// SIMATIC STEP 7 (V5.x) project Kukla-DP-DWC7A
// CPU: CPU 315-2 PN/DP
// station: Hardware
// station: SIMATIC 300(1)
// station: P_ADR_BUS
// program: S7 Prog DWC7A

SYMBOL_TABLE
"CMD_KSW"	DB 40	DB 40
"ACT_KSW"	DB 41	DB 41	// Datablock for Continious weighing system 1
"COMM_KSW7"	FC 40	FC 40
"PLC_toKSW7B"	VAT 1		// DB40_PLC_to_KSW
"KSW7B_to_PLC"	VAT 2		// DB41_KSW7_to_PLC
END_SYMBOL_TABLE

TYPE UDT 400
VERSION : 1.0
  STRUCT
   bWCx_Warning : BOOL ;	// 24: Warnung
   bWCx_RdyToOperate : BOOL ;	// 25: Betriebsbereit
   bWCx_XD0 : BOOL ;	// 26:
   bWCx_XD1 : BOOL ;	// 27:
   bWCx_XD2 : BOOL ;	// 28:
   bWCx_XD3 : BOOL ;	// 29:
   bWCx_Crtl_30 : BOOL ;	// 30: ---
   bWCx_FieldRelais4 : BOOL ;	// 31: Fieldrelais 4
   bWCx_DriveBolcked : BOOL ;	// 16: Antriebe gesperrt
   bWCx_EmcyStopActiv : BOOL ;	// 17: Notaus aktiv
   bWCx_MainDriveRuns : BOOL ;	// 18: Läuft
   bWCx_MainDriveJog : BOOL ;	// 19: Hauptantrieb JOG
   bWCx_FieldRelais0 : BOOL ;	// 20: Fieldrelais 0
   bWCx_FieldRelais1 : BOOL ;	// 21: Fieldrelais 1
   bWCx_FieldRelais2 : BOOL ;	// 22: Fieldrelais 2
   bWCx_FieldRelais3 : BOOL ;	// 23: Fieldrelais 3
   bWCx_BinMaxLevel : BOOL ;	// 08: Max Meldung
   bWCx_BinMaxMaxLevel : BOOL ;	// 09: Max Max Meldung
   bWCx_BatchWeightFault : BOOL ;	// 10: Mengenfehler
   bWCx_Crtl_11 : BOOL ;	// 11: ---
   bWCx_Crtl_12 : BOOL ;	// 12: ---
   bWCx_Crtl_13 : BOOL ;	// 13: ---
   bWCx_ProdRelease : BOOL ;	// 14: Materialfreigabe
   bWCx_Remote : BOOL ;	// 15: Remote
   bWCx_Crtl_00 : BOOL ;	// 00: ---
   bWCx_StartBatch : BOOL ;	// 01: Charge Start
   bWCx_BatchCoarseStream : BOOL ;	// 02: Charge Grobstrom
   bWCx_BatchFineStream : BOOL ;	// 03: Charge Feinstrom
   bWCx_ReFillingOn : BOOL ;	// 04: Füllen ein
   bWCx_BinEmpty : BOOL ;	// 05: Leer
   bWCx_BinMinMinLevel : BOOL ;	// 06: Min Min Meldung
   bWCx_BinMinLevel : BOOL ;	// 07: Min Meldung
  END_STRUCT ;	
END_TYPE

TYPE UDT 420
VERSION : 1.0
  STRUCT
   bWCx_Cmd_FieldOpto4 : BOOL ;	// 24: Feldopto 4
   bWCx_Cmd_DriveFault : BOOL ;	// 25: Motorstoerung
   bWCx_Cmd_26 : BOOL ;	// 26: ---
   bWCx_Cmd_27 : BOOL ;	// 27: ---
   bWCx_Cmd_28 : BOOL ;	// 28: ---
   bWCx_Cmd_29 : BOOL ;	// 29: ---
   bWCx_Cmd_30 : BOOL ;	// 30: ---
   bWCx_Cmd_31 : BOOL ;	// 31: ---
   bWCx_Cmd_BlockDrive : BOOL ;	// 16: Antriebsperre
   bWCx_Cmd_EmcyStop : BOOL ;	// 17: Notaus is aktiv
   bWCx_Cmd_DriveIsRuning : BOOL ;	// 18: Antrieb läuft Status
   bWCx_Cmd_DriveJog : BOOL ;	// 19: Antrieb Jog aktivieren
   bWCx_Cmd_FieldOpto0 : BOOL ;	// 20: Feldopto 0
   bWCx_Cmd_FieldOpto1 : BOOL ;	// 21: Feldopto 1
   bWCx_Cmd_FieldOpto2 : BOOL ;	// 22: Feldopto 2
   bWCx_Cmd_FieldOpto3 : BOOL ;	// 23: Feldopto 3
   bWCx_Cmd_08 : BOOL ;	// 08: ---
   bWCx_Cmd_StartBatch : BOOL ;	// 09: Charge starten
   bWCx_Cmd_InterruptBatch : BOOL ;	// 10: Charge unterbrechen
   bWCx_Cmd_CancelBatch : BOOL ;	// 11: Charge abbrechen
   bWCx_Cmd_FineStream : BOOL ;	// 12: Feinstrom erzwingen
   bWCx_Cmd_Emtying : BOOL ;	// 13: System entleeren
   bWCx_Cmd_14 : BOOL ;	// 14: ---
   bWCx_Cmd_Remote : BOOL ;	// 15: Remote aktivieren
   bWCx_Cmd_00 : BOOL ;	// 00: ---
   bWCx_Cmd_SetZero : BOOL ;	// 01: Nullpunkt setzen <0> STARTEN
   bWCx_Cmd_StartTare : BOOL ;	// 02: Tarierung starten
   bWCx_Cmd_ClrCounterB : BOOL ;	// 03: Zähler B zurücksetzen
   bWCx_Cmd_MaxMaxSensor : BOOL ;	// 04: Max Max Sensoreingang
   bWCx_Cmd_MaxSensor : BOOL ;	// 05: Max Sensoreingang
   bWCx_Cmd_MinSensor : BOOL ;	// 06: Min Sensoreingang
   bWCx_Cmd_MinMinSensor : BOOL ;	// 07: Min Min Sensoreingang
  END_STRUCT ;	
END_TYPE

FUNCTION "COMM_KSW7" : VOID	// FC 40
TITLE = <DWC-7A / KUKLA DataExchange>
//KNOW_HOW_PROTECT 
//
AUTHOR : Ratzi
FAMILY : com_dwc7
NAME : fc_7A
VERSION : 1.0
VAR_INPUT
  P97200_BusInDW00 : DINT ;	// SetValue DW00 to KSW-7
  P97201_BusInDW04 : DINT ;	// SetValue DW04 to KSW-7
  P97202_BusInDW08 : DINT ;	// SetValue DW08 to KSW-7
  P97203_BusInDW12 : DINT ;	// SetValue DW12 to KSW-7
  P97204_BusInDW16 : DINT ;	// SetValue DW16 to KSW-7
  P97205_BusInDW20 : DINT ;	// SetValue DW20 to KSW-7
  P97206_BusInDW24 : DINT ;	// SetValue DW24 to KSW-7
  P97207_BusInDW28 : DINT ;	// SetValue DW28 to KSW-7
  Adr_In : INT ;	// HW-Manager Eingang/Input Area Baseaddress
  Adr_Out : INT ;	// HW-Manager Ausgang/Qutput Area Baseaddress
END_VAR
VAR_OUTPUT
  P97400_BusOutDW00 : DINT ;	// ProcessValue DW00 from KSW-7
  P97401_BusOutDW04 : DINT ;	// ProcessValue DW04 from KSW-7
  P97402_BusOutDW08 : DINT ;	// ProcessValue DW08 from KSW-7
  P97403_BusOutDW12 : DINT ;	// ProcessValue DW12 from KSW-7
  P97404_BusOutDW16 : DINT ;	// ProcessValue DW16 from KSW-7
  P97405_BusOutDW20 : DINT ;	// ProcessValue DW20 from KSW-7
  P97406_BusOutDW24 : DINT ;	// ProcessValue DW24 from KSW-7
  P97407_BusOutDW28 : DINT ;	// ProcessValue DW28 from KSW-7
  P97408_BusOutDW32 : DINT ;	// ProcessValue DW32 from KSW-7
  P97409_BusOutDW36 : DINT ;	// ProcessValue DW36 from KSW-7
  P97410_BusOutDW40 : DINT ;	// ProcessValue DW40 from KSW-7
  P97411_BusOutDW44 : DINT ;	// ProcessValue DW44 from KSW-7
  P97412_BusOutDW48 : DINT ;	// ProcessValue DW48 from KSW-7
  P97413_BusOutDW52 : DINT ;	// ProcessValue DW52 from KSW-7
  P97414_BusOutDW56 : DINT ;	// ProcessValue DW56 from KSW-7
  P97415_BusOutDW60 : DINT ;	// ProcessValue DW60 from KSW-7
  bOnline : BOOL ;	// DWC-7 online signal
END_VAR
BEGIN
NETWORK
TITLE =    <Read Set-Values to DWC-7>
      LAR1  P#P 0.0;
      L     #Adr_Out;
      SLW   3;
      +AR1;
      L     #P97200_BusInDW00;
      T     D [AR1,P#0.0];
      L     #P97201_BusInDW04;
      T     D [AR1,P#4.0];
      L     #P97202_BusInDW08;
      T     D [AR1,P#8.0];
      L     #P97203_BusInDW12;
      T     D [AR1,P#12.0];
      L     #P97204_BusInDW16;
      T     D [AR1,P#16.0];
      L     #P97205_BusInDW20;
      T     D [AR1,P#20.0];
      L     #P97206_BusInDW24;
      T     D [AR1,P#24.0];
      L     #P97207_BusInDW28;
      T     D [AR1,P#28.0];
NETWORK
TITLE =    <Write current-Values to DWC-7>
      LAR1  P#P 0.0;
      L     #Adr_In;
      SLW   3;
      +AR1;
      L     D [AR1,P#0.0];
      T     #P97400_BusOutDW00;
      L     D [AR1,P#4.0];
      T     #P97401_BusOutDW04;
      L     D [AR1,P#8.0];
      T     #P97402_BusOutDW08;
      L     D [AR1,P#12.0];
      T     #P97403_BusOutDW12;
      L     D [AR1,P#16.0];
      T     #P97404_BusOutDW16;
      L     D [AR1,P#20.0];
      T     #P97405_BusOutDW20;
      L     D [AR1,P#24.0];
      T     #P97406_BusOutDW24;
      L     D [AR1,P#28.0];
      T     #P97407_BusOutDW28;
      L     D [AR1,P#32.0];
      T     #P97408_BusOutDW32;
      L     D [AR1,P#36.0];
      T     #P97409_BusOutDW36;
      L     D [AR1,P#40.0];
      T     #P97410_BusOutDW40;
      L     D [AR1,P#44.0];
      T     #P97411_BusOutDW44;
      L     D [AR1,P#48.0];
      T     #P97412_BusOutDW48;
      L     D [AR1,P#52.0];
      T     #P97413_BusOutDW52;
      L     D [AR1,P#56.0];
      T     #P97414_BusOutDW56;
      L     D [AR1,P#60.0];
      T     #P97415_BusOutDW60;
NETWORK
TITLE =    <Process Online by all Numbers unequal 0>
      A     #bOnline;
      AN    #bOnline;
      =     #bOnline;
      L     #P97400_BusOutDW00;
      L     L#0;
      <>D;
      O     #bOnline;
      =     #bOnline;
      L     #P97401_BusOutDW04;
      L     L#0;
      <>D;
      O     #bOnline;
      =     #bOnline;
      L     #P97402_BusOutDW08;
      L     L#0;
      <>D;
      O     #bOnline;
      =     #bOnline;
      L     #P97403_BusOutDW12;
      L     L#0;
      <>D;
      O     #bOnline;
      =     #bOnline;
      L     #P97404_BusOutDW16;
      L     L#0;
      <>D;
      O     #bOnline;
      =     #bOnline;
      L     #P97405_BusOutDW20;
      L     L#0;
      <>D;
      O     #bOnline;
      =     #bOnline;
      L     #P97406_BusOutDW24;
      L     L#0;
      <>D;
      O     #bOnline;
      =     #bOnline;
      L     #P97407_BusOutDW28;
      L     L#0;
      <>D;
      O     #bOnline;
      =     #bOnline;
      L     #P97408_BusOutDW32;
      L     L#0;
      <>D;
      O     #bOnline;
      =     #bOnline;
      L     #P97409_BusOutDW36;
      L     L#0;
      <>D;
      O     #bOnline;
      =     #bOnline;
      L     #P97410_BusOutDW40;
      L     L#0;
      <>D;
      O     #bOnline;
      =     #bOnline;
      L     #P97411_BusOutDW44;
      L     L#0;
      <>D;
      O     #bOnline;
      =     #bOnline;
      L     #P97412_BusOutDW48;
      L     L#0;
      <>D;
      O     #bOnline;
      =     #bOnline;
      L     #P97413_BusOutDW52;
      L     L#0;
      <>D;
      O     #bOnline;
      =     #bOnline;
      L     #P97414_BusOutDW56;
      L     L#0;
      <>D;
      O     #bOnline;
      =     #bOnline;
      L     #P97415_BusOutDW60;
      L     L#0;
      <>D;
      O     #bOnline;
      =     #bOnline;
END_FUNCTION

DATA_BLOCK "CMD_KSW"	// DB 40
VERSION : 0.0
  STRUCT
   KSW7_SET_DW00 : UDT 420;	// P97200 BusIn DW00 - 01:WC00 CMD
   KSW7_SET_DW04 : DINT ;	// P97201 BusIn DW04 - 10: Bus 1 ABS
   KSW7_SET_DW08 : UDT 420;	// P97202 BusIn DW08 - 01:WC10 CMD
   KSW7_SET_DW12 : DINT ;	// P97203 BusIn DW12 - 11: Bus 2 ABS
   KSW7_SET_DW16 : UDT 420;	// P97204 BusIn DW16 - 01:WC20 CMD
   KSW7_SET_DW20 : DINT ;	// P97205 BusIn DW20 - 12: Bus 3 ABS
   KSW7_SET_DW24 : DINT ;	// P97206 BusIn DW24 - 00: ---
   KSW7_SET_DW28 : DINT ;	// P97207 BusIn DW28 - 00: ---
  END_STRUCT ;	
BEGIN
END_DATA_BLOCK

DATA_BLOCK "ACT_KSW"	// DB 41
VERSION : 0.0
  STRUCT
   KSW7_ACT_DW00 : UDT 400;	// P97400 BusOut DW00 - 28: WC00 Controlbits 1
   KSW7_ACT_DW04 : DINT ;	// P97401 BusOut DW04 - 10: WC00 Abs
   KSW7_ACT_DW08 : DINT ;	// P97402 BusOut DW08 - 55: WC00 Istcharge
   KSW7_ACT_DW12 : DINT ;	// P97403 BusOut DW12 - 37: WC00 Dosiersollwert
   KSW7_ACT_DW16 : DINT ;	// P97404 BusOut DW16 - 46: WC00 Chargenschritt
   KSW7_ACT_DW20 : UDT 400;	// P97405 BusOut DW20 - 29: WC10 Controlbits 1
   KSW7_ACT_DW24 : DINT ;	// P97406 BusOut DW24 - 11: WC10 Abs
   KSW7_ACT_DW28 : DINT ;	// P97407 BusOut DW28 - 56: WC10 Istcharge
   KSW7_ACT_DW32 : DINT ;	// P97408 BusOut DW32 - 38: WC10 Dosiersollwert
   KSW7_ACT_DW36 : DINT ;	// P97409 BusOut DW36 - 47: WC10 Chargenschritt
   KSW7_ACT_DW40 : UDT 400;	// P97410 BusOut DW40 - 30: WC20 Controlbits 1
   KSW7_ACT_DW44 : DINT ;	// P97411 BusOut DW44 - 12: WC20 Abs
   KSW7_ACT_DW48 : DINT ;	// P97412 BusOut DW48 - 57: WC20 Istcharge
   KSW7_ACT_DW52 : DINT ;	// P97413 BusOut DW52 - 39: WC20 Dosiersollwert
   KSW7_ACT_DW56 : DINT ;	// P97414 BusOut DW56 - 48: WC20 Chargenschritt
   KSW7_ACT_DW60 : DINT ;	// P97415 BusOut DW60 - 00: ---
   KSW7_ACT_DW64 : DINT ;	// P97416 BusOut DW64 - 00: ---
   KSW7_ACT_DW68 : DINT ;	// P97417 BusOut DW68 - 00: ---
   KSW7_ACT_DW72 : DINT ;	// P97418 BusOut DW72 - 00: ---
   KSW7_ACT_DW76 : DINT ;	// P97419 BusOut DW76 - 00: ---
  END_STRUCT ;	
BEGIN
END_DATA_BLOCK

ORGANIZATION_BLOCK OB 1
TITLE = "Main Program Sweep (Cycle)"
VERSION : 0.1
VAR_TEMP
  OB1_EV_CLASS : BYTE ;	//Bits 0-3 = 1 (Coming event), Bits 4-7 = 1 (Event class 1)
  OB1_SCAN_1 : BYTE ;	//1 (Cold restart scan 1 of OB 1), 3 (Scan 2-n of OB 1)
  OB1_PRIORITY : BYTE ;	//Priority of OB Execution
  OB1_OB_NUMBR : BYTE ;	//1 (Organization block 1, OB1)
  OB1_RESERVED_1 : BYTE ;	//Reserved for system
  OB1_RESERVED_2 : BYTE ;	//Reserved for system
  OB1_PREV_CYCLE : INT ;	//Cycle time of previous OB1 scan (milliseconds)
  OB1_MIN_CYCLE : INT ;	//Minimum cycle time of OB1 (milliseconds)
  OB1_MAX_CYCLE : INT ;	//Maximum cycle time of OB1 (milliseconds)
  OB1_DATE_TIME : DATE_AND_TIME ;	//Date and time OB1 started
END_VAR
BEGIN
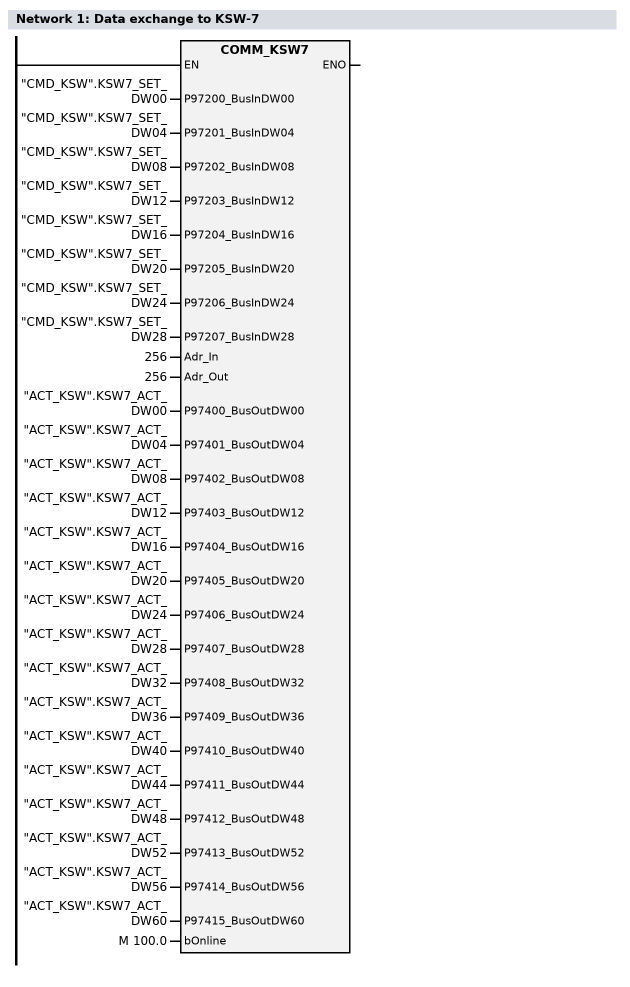
NETWORK
TITLE = Data exchange to KSW-7 
      CALL  "COMM_KSW7" (
           P97200_BusInDW00         := "CMD_KSW".KSW7_SET_DW00,
           P97201_BusInDW04         := "CMD_KSW".KSW7_SET_DW04,
           P97202_BusInDW08         := "CMD_KSW".KSW7_SET_DW08,
           P97203_BusInDW12         := "CMD_KSW".KSW7_SET_DW12,
           P97204_BusInDW16         := "CMD_KSW".KSW7_SET_DW16,
           P97205_BusInDW20         := "CMD_KSW".KSW7_SET_DW20,
           P97206_BusInDW24         := "CMD_KSW".KSW7_SET_DW24,
           P97207_BusInDW28         := "CMD_KSW".KSW7_SET_DW28,
           Adr_In                   := 256,
           Adr_Out                  := 256,
           P97400_BusOutDW00        := "ACT_KSW".KSW7_ACT_DW00,
           P97401_BusOutDW04        := "ACT_KSW".KSW7_ACT_DW04,
           P97402_BusOutDW08        := "ACT_KSW".KSW7_ACT_DW08,
           P97403_BusOutDW12        := "ACT_KSW".KSW7_ACT_DW12,
           P97404_BusOutDW16        := "ACT_KSW".KSW7_ACT_DW16,
           P97405_BusOutDW20        := "ACT_KSW".KSW7_ACT_DW20,
           P97406_BusOutDW24        := "ACT_KSW".KSW7_ACT_DW24,
           P97407_BusOutDW28        := "ACT_KSW".KSW7_ACT_DW28,
           P97408_BusOutDW32        := "ACT_KSW".KSW7_ACT_DW32,
           P97409_BusOutDW36        := "ACT_KSW".KSW7_ACT_DW36,
           P97410_BusOutDW40        := "ACT_KSW".KSW7_ACT_DW40,
           P97411_BusOutDW44        := "ACT_KSW".KSW7_ACT_DW44,
           P97412_BusOutDW48        := "ACT_KSW".KSW7_ACT_DW48,
           P97413_BusOutDW52        := "ACT_KSW".KSW7_ACT_DW52,
           P97414_BusOutDW56        := "ACT_KSW".KSW7_ACT_DW56,
           P97415_BusOutDW60        := "ACT_KSW".KSW7_ACT_DW60,
           bOnline                  := M 100.0);
      NOP   0;
END_ORGANIZATION_BLOCK
